TYPE DeviceLabel :
STRUCT

	//Structure contains all field data on a device label,
	//There are 4 fields in total, unclear what each field is	

	SN : STRING(30);	//Electronic Serial Number
	SKU : STRING(30);	//OEM SKU
	MSN : STRING(30);	//Material Serial Number
	PPN : STRING(30);	//Product part number (Apple only)
	cERROR : STRING(30) := 'ERROR';
	
END_STRUCT
END_TYPE

(* stored: Version 1.1.0.1, ProductVersion 3.1.4024.6
   DUT DeviceLabel: Id {ed2cea86-ee82-410b-859d-c5e68cc52030} *)
